FUNCTION_BLOCK OR_BOOL (* IEC 61131-3 Boolean OR *)
  (* Standard: 61131-3 *)
  (* Version 0.1, 2006-09-07, JHC, Holobloc Inc, Converted to Template *)
  (* Version 0.0, 2004-12-15, JHC, Rockwell Automation, Converted from SRC format. *)
  (* Compiler header: package fb.rt.plc.bits; *)
  (* Compiler classdef: (i1 || i2) *)
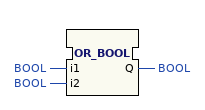
  VAR_INPUT
    i1 : BOOL;
    i2 : BOOL;
  END_VAR
  VAR_OUTPUT
    Q : BOOL;
  END_VAR
END_FUNCTION_BLOCK
